FUNCTION_BLOCK GEN_RMP (* this signal generator generates a ramp wave output *)
  (* Standard: 61499-1; Description: version 1.4	10. mar. 2009 programmer 	oscat tested BY		oscat this signal generator generates a ramp wave output. The ramp wave signal is defined by period time (PT), amplitude (AM), offset (OS) and a specific delay for the output signal (DL). The Output waveform will have its minimum peak at OS and its maximum peak at AM + OS. The delay input can delay a signal up to PT, this can be useful to synchronize different generators and generate interleaving signals. in addition to the analog output Out there is a second boolean output Q with is true for one cycle when the ramp starts. *)
  (* Version 1.0, 2025-12-21, Franz Höpfinger, initial API and implementation and/or initial documentation *)
  PACKAGE OSCAT::Basic::POUs::Engineering::signal_generators;
  IMPORT OSCAT::Basic::POUs::Mathematical::MODR;
  IMPORT OSCAT::Basic::POUs::Mathematical::FRACT;
  IMPORT OSCAT::Basic::POUs::conversion::TIME_TO_REAL;
  IMPORT OSCAT::Basic::POUs::Time_Date::MULTIME;
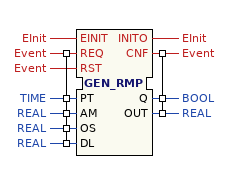
  EVENT_INPUT
    EINIT : EInit; (* Init Request *)
    REQ WITH PT, AM, OS, DL; (* Normal Execution Request *)
    RST; (* Reset *)
  END_EVENT
  EVENT_OUTPUT
    INITO : EInit; (* Init Confirmation *)
    CNF WITH Q, OUT; (* Execution Confirmation *)
  END_EVENT
  VAR_INPUT
    PT : TIME := T#1s; (* Period Time *)
    AM : REAL := 1.0; (* Amplitude *)
    OS : REAL; (* Offset *)
    DL : REAL; (* Delay *)
  END_VAR
  VAR_OUTPUT
    Q : BOOL; (* Pulse Output *)
    OUT : REAL; (* Ramp Output *)
  END_VAR
  VAR
    tx : TIME;
    last : TIME;
    init : BOOL;
    temp : REAL;
    ltemp : REAL;
    DL_M : REAL;
  END_VAR
  EC_STATES
    EINIT : EINIT -> INITO;
    REQ : REQ -> CNF;
    RST : RST -> CNF;
  END_STATES
  ALGORITHM EINIT IN ST:
init := FALSE;
  END_ALGORITHM
  ALGORITHM RST IN ST:
init := TRUE;
last := tx;
tx := T#0s;
  END_ALGORITHM
  ALGORITHM REQ IN ST:
(* read system time and prepare input data *)
tx := NOW_MONOTONIC() - last;
DL_M := MODR(DL, 1.0);
IF DL_M < 0.0 THEN
	DL_M := 1.0 - DL_M;
END_IF;

(* init section *)
IF NOT init THEN
	this.RST();
END_IF;

(* add last if one cycle is finished *)
IF tx >= PT THEN
	last := last + PT;
	tx := tx - PT;
END_IF;

(* generate sine wave *)
ltemp := temp;
IF PT > T#0s THEN
	temp := FRACT(TIME_TO_REAL(tx + MULTIME(PT, DL_M)) / TIME_TO_REAL(PT));
END_IF;
OUT := AM * temp + OS;

(* boolean output Q *)
Q := temp < ltemp;
  END_ALGORITHM
END_FUNCTION_BLOCK
